// Returns whether or not all the data before the limit has been read.
FUNCTION INTERNAL F_SbhIsReachedLimit : BOOL
VAR_IN_OUT
    stState     : ST_ParserInternalState;
END_VAR
VAR
    nCurrentAbsolutPos : UDINT;
END_VAR


IF stState.nCurrentLimit = TO_UDINT(-1) THEN
    RETURN;
END_IF

nCurrentAbsolutPos := stState.nTotalBytesRetired + stState.nBufferPos;
F_SbhIsReachedLimit := nCurrentAbsolutPos >= stState.nCurrentLimit;

END_FUNCTION

(* stored: Version 1.1.0.1
   POU F_SbhIsReachedLimit: Id {28c6146d-a251-4e02-a457-09194433aa7a}, SpecialFunc None *)
